FUNCTION_BLOCK Test_TStreamAdd_Read_INT EXTENDS T_UnitTestBase
VAR
    Stream : T_Stream(StreamLength := 2);
END_VAR



Stream.Init(2);

Stream.Add_INT(1234);
    
Assertion.AssertEquals_UDINT(
    Expected := 2,
    Actual := Stream.Position,
    VariableName := 'Stream.Position');
    
Stream.Seek(0);

Assertion.AssertEquals_INT(
    Expected := 1234,
    Actual := Stream.Read_INT(),
    VariableName := 'Stream.Read_INT()');
    
Assertion.AssertEquals_UDINT(
    Expected := 2,
    Actual := Stream.Position,
    VariableName := 'Stream.Position');
    
    
TestFinished();

END_FUNCTION_BLOCK

(* stored: Version 1.1.0.1, ProductVersion 3.1.4024.4
   POU Test_TStreamAdd_Read_INT: Id {76a55d7b-1486-4a4a-82f7-72fd80dc368a}, SpecialFunc None *)
